// TIA Portal project "Motor ansteuern(ohne Geber)_V18" (V18)

(* hardware
DEVICE "S71500/ET200MP-Station_2"  S7-1500 station
   slot 0: "Profilschiene_0"  Rack  6ES7 590-1***0-0AA0
   slot 1: "PLC_2"  CPU 1513-1 PN  6ES7 513-1AL02-0AB0  V2.8
      slot 3: "CPU-Display_1"  6ES7591-1AA00-0AA0
      slot 32768: "PROFINET-Schnittstelle_1"  X1
         slot 32769: "Port_1"  X1 P1
         slot 32770: "Port_2"  X1 P2
      slot 34817: "Virtual CP interface port_1"  Virtual CP interface port  Virtual CP interface port
   slot 2: "DQ 16x24VDC/0.5A HF_1"  DQ 16x24VDC/0.5A HF  6ES7 522-1BH01-0AB0  V1.1
   slot 3: "TM PTO 4"  TM PTO 4  6ES7 553-1AA00-0AB0  V1.0
   slot 4: "TM PTO 4_1"  TM PTO 4  6ES7 553-1AA00-0AB0  V1.0
*)

// ===== PLC "PLC_2"  CPU 1513-1 PN =====

VAR_GLOBAL   // PLC tag table "Standard-Variablentabelle"
   "PositioningAxis_1_Actor_Interface_AddressIn" AT %I0.0 : "PD_TEL3_IN";
   "PositioningAxis_1_Actor_Interface_AddressOut" AT %Q0.0 : "PD_TEL3_OUT";
END_VAR

DATA_BLOCK "SpeedAxis_1"   // DB1, Motion_DB
{ S7_Optimized_Access := 'TRUE' }
AUTHOR : SIMATIC
FAMILY : MC_1500
VERSION : 5.0
// stored: InstanceOfName TO_SpeedAxis
"TO_SpeedAxis"
BEGIN
END_DATA_BLOCK

ORGANIZATION_BLOCK "Main"   // OB1, FBD, ProgramCycle
TITLE = "Main Program Sweep (Cycle)"
{ S7_Optimized_Access := 'TRUE' }
VERSION : 0.1
   VAR_INPUT
      Initial_Call : Bool;   // Initial call of this OB
      Remanence : Bool;   // =True, if remanent data are available
   END_VAR
BEGIN

REGION Network 1
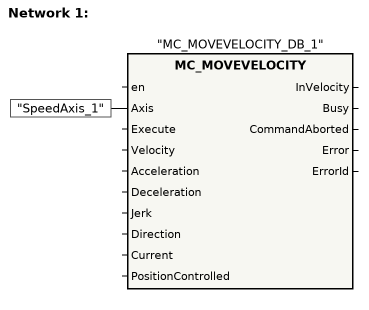
   "MC_MOVEVELOCITY_DB_1"(Axis := "SpeedAxis_1");   // MC_MOVEVELOCITY
END_REGION
END_ORGANIZATION_BLOCK